ABB RAPID module: Calib_t_HSLU_GripperZimmer1.modx

MODULE Calib_t_HSLU_GripperZimmer1(READONLY)
 LOCAL CONST string dataName := "t_HSLU_GripperZimmer1";
 LOCAL CONST string mechUnitRef := "ROB_1";
 LOCAL CONST string toolRef := "tool0";
 LOCAL CONST robtarget pTCP_Point1 := [[898.9413,-265.559,255.0308],[0.03146343,-0.6501036,0.7215203,0.236186],[-1,0,-2,0],[8.999999E+09,8.999999E+09,8.999999E+09,8.999999E+09,8.999999E+09,8.999999E+09]];
 LOCAL CONST robtarget pTCP_Point2 := [[777.0348,-251.7125,239.3385],[0.2762992,-0.2379081,0.9226829,0.1253589],[-1,1,-2,0],[8.999999E+09,8.999999E+09,8.999999E+09,8.999999E+09,8.999999E+09,8.999999E+09]];
 LOCAL CONST robtarget pTCP_Point3 := [[954.6644,-161.6835,241.3231],[0.2340333,0.8343173,-0.4532449,-0.2090746],[-1,-1,-2,0],[8.999999E+09,8.999999E+09,8.999999E+09,8.999999E+09,8.999999E+09,8.999999E+09]];
 !------------------------------------------------------------------------------
 !<auto-generated>
 !This code was generated by a tool.

 !<auto-generated>
 !Changes to this file may cause incorrect behavior and will be lost if
 !the code is regenerated.
 !</auto-generated>
 !------------------------------------------------------------------------------



 ! 06 May 2026 20:16:42 by Default User from ABB Robotics FlexPendant
 ! Old Value: [TRUE,[[0,0,189],[0.707107,0,0,0.707107]],[3,[0,0,4],[1,0,0,0],0,0,0]]
 ! Maxerror, Minerror, Meanerror Values: 0, 0, 0


ENDMODULE
